// TIA Portal V16 export
// export: Created 2021-07-12T14:47:17.9978972Z, ExportSetting WithDefaults, DisplayName Totally Integrated Automation Portal, DisplayVersion V16, DisplayName TIA Portal Version Control Interface, DisplayVersion V16, DisplayName TIA Portal Openness, DisplayVersion V16, DisplayName STEP 7 Professional, DisplayVersion V16, DisplayName STEP 7 Safety, DisplayVersion V16, DisplayName WinCC Professional, DisplayVersion V16
TYPE "SimaHydTO_typeHMIConnectionAdvancedAxisControl"
TITLE = SimaHydTO_typeHMIConnectionAdvancedAxisControl
// HMI interface: Advanced axis control
// stored: IsFailsafeCompliant false
   STRUCT
      Command { S7_SetPoint := 'True'} : "SimaHydTO_typeHMIConnectionAdvancedAxisControlCommand";   // Command (HMI -> PLC)
      Status { S7_SetPoint := 'True'} : "SimaHydTO_typeHMIConnectionAdvancedAxisControlStatus";   // Status (PLC -> HMI)
   END_STRUCT;
END_TYPE
